// TIA Portal V19 export
FUNCTION "FC_TechScan" : Void   // FC42, STL
TITLE = Initialisieren Technologische Parameter
{ S7_Optimized_Access := 'FALSE' }
// stored: AutoNumber false
   VAR_INPUT
      WT_DB_Nr : Int;
   END_VAR
   VAR_TEMP
      WT_DB : Word;
      lastCmd : Int;
      Count : Int;
      AdrReg1 : DWord;
      AdrReg2 : DWord;
      typTaktzeit : Int;
      Expo : DInt;
   END_VAR
BEGIN

NETWORK
TITLE = Bereichstakte Beladestand 1 laden

//-------------------------------
//WT-DB öffnen und Adressregister
//retten
//-------------------------------
      TAR1;
      T     #AdrReg1;
      TAR2;
      T     #AdrReg2;

      L     "DB_ANLAGE".config.Taktzeit_typ;
      T     #typTaktzeit;

      L     #WT_DB_Nr;
      T     #WT_DB;
      OPN   DB [#WT_DB];

//-------------------------------
//Initialisieren Kopfdaten
//-------------------------------
      L     0;
      T     %DBB54;  //"DB_WT1".Variante0//Bereichstakte
      T     %DBB55;  //"DB_WT1".Variante1  Technologie 0=Natur, 1=Matt, 2=Glänzen
      T     %DBB56;  //"DB_WT1".Variante2  Farbe 0-6
      T     %DBB57;  //"DB_WT1".Variante3  Beizzeit 0=<60s 1=<8min 2=>8min
      T     %DBB58;  //"DB_WT1".Variante4  Glänzzeit 0=kurz 1=mittel 2=lang
      T     %DBB59;  //"DB_WT1".Variante5


NETWORK
TITLE = Scan Technologie
//-------------------------------
//Scan von Befehl 0 bis Anzahl
//-------------------------------
      L     %DBW0;  //"DB_WT1".ANZAHL
      T     #lastCmd;
      L     0;
retC: T     #Count;
      L     #lastCmd;
      >=I;
      JC    Ende;

      L     #Count;
      L     %DBW4;  //"DB_WT1".LENG
      *I;
      L     %DBW2;  //"DB_WT1".OFFSET
      +I;
      SLD   3;
      LAR1;
      OPN   DB [#WT_DB];
      L     DBB [AR1, P#0.0];  //CmdID
      L     0;
      ==I;
      JC    Ende;

nexC: L     #Count;
      +     1;
      JU    retC;

NETWORK
TITLE = Parameter abfregen und laden

NETWORK
TITLE = Ende Scandurchlauf
Ende: L     #AdrReg1;
      LAR1;
      L     #AdrReg2;
      LAR2;
      BE;
END_FUNCTION
